(* IEC 61131-3 sources: plc-vscode/tests/st/test-ready/trust-platform/examples/vendor_library_stubs/src, 2 files *)

(* ---- Configuration.st ---- *)
CONFIGURATION VendorStubsDemo
RESOURCE Cpu0 ON PLC
    TASK MainTask (INTERVAL := T#100ms, PRIORITY := 1);
    PROGRAM Main WITH MainTask : Main;
END_RESOURCE
END_CONFIGURATION

(* ---- Main.st ---- *)
PROGRAM Main
VAR
    Connect : TCON;
    Normalizer : NORM_X;
    Scaler : SCALE_X;
    Request : BOOL := TRUE;
    RawInput : REAL := 42.0;
    Percent : REAL;
    Engineering : REAL;
END_VAR

Connect(REQ := Request);
Normalizer(X := RawInput, X_MIN := 0.0, X_MAX := 100.0, Y => Percent);
Scaler(
    X := Percent,
    X_MIN := 0.0,
    X_MAX := 1.0,
    Y_MIN := 0.0,
    Y_MAX := 1000.0,
    Y => Engineering
);
END_PROGRAM
